PROGRAM MAIN
VAR
	// Histeres da temperatura definida
	Histerese 		: REAL := 1;
	LigaCompressor 	: SR;
	
END_VAR

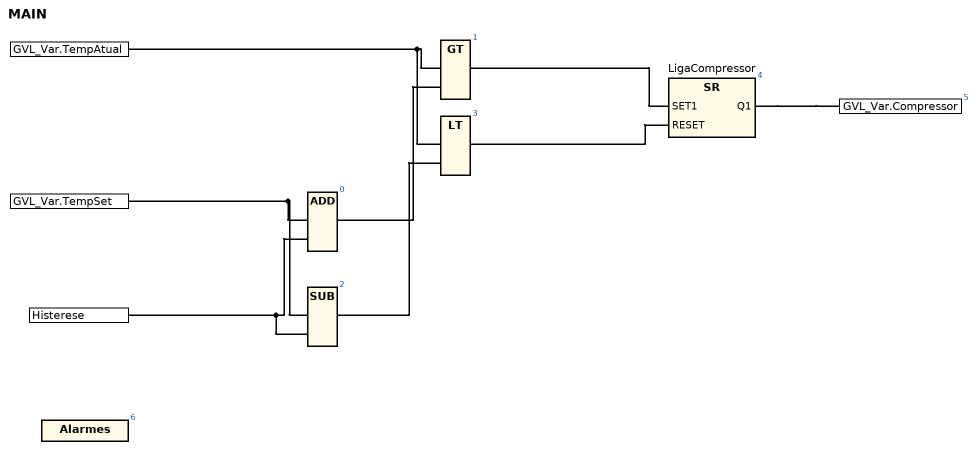
LigaCompressor(SET1 := GVL_Var.TempAtual > GVL_Var.TempSet + Histerese, RESET := GVL_Var.TempAtual < GVL_Var.TempSet - Histerese); // SR
GVL_Var.Compressor := LigaCompressor.Q1;
Alarmes();

END_PROGRAM

(* stored: Version 1.1.0.1
   POU MAIN: Id {9326eecf-71cc-4138-9994-23fc16f5e55a}, SpecialFunc None *)
